FUNCTION_BLOCK SFC4 (* Basic Function Block Type *)
  (* Standard: 61499-2 *)
  (* Version 0.2, 2003-12-04, JHC, Rockwell Automation, Renamed for better indexing. *)
  (* Version 0.1, 2002-11-05, JHC, Rockwell Automation, Corrected missing ST element in Algorithm REQ. *)
  (* Version 0.0, 2000-05-30, JHC, Rockwell Automation *)
  (* Compiler header: package fb.rt.pnp; *)
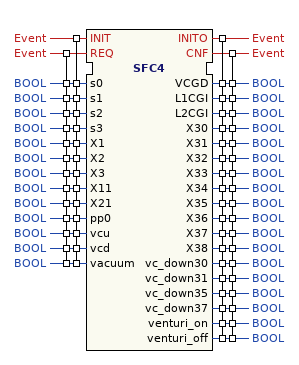
  EVENT_INPUT
    INIT WITH s0, s0, s0, s1, s2, s3, X1, X2, X3, X11, X21, pp0, vcu, vcd, vacuum; (* Initialization Request *)
    REQ WITH s0, s0, s1, s2, s3, X1, X2, X3, X11, X21, pp0, vcu, vcd, vacuum; (* Normal Execution Request *)
  END_EVENT
  EVENT_OUTPUT
    INITO WITH VCGD, L1CGI, L2CGI, X30, X30, X31, X32, X33, X34, X35, X36, X37, X38, vc_down30, vc_down31, vc_down35, vc_down37, venturi_on, venturi_off; (* Initialization Confirm *)
    CNF WITH VCGD, L1CGI, L2CGI, X30, X30, X31, X32, X33, X34, X35, X36, X37, X38, vc_down30, vc_down31, vc_down35, vc_down37, venturi_on, venturi_off; (* Execution Confirmation *)
  END_EVENT
  VAR_INPUT
    s0 : BOOL; (* Input event qualifier *)
    s1 : BOOL; (* Input event qualifier *)
    s2 : BOOL; (* Input event qualifier *)
    s3 : BOOL; (* Input event qualifier *)
    X1 : BOOL; (* Input event qualifier *)
    X2 : BOOL; (* Input event qualifier *)
    X3 : BOOL; (* Input event qualifier *)
    X11 : BOOL; (* Input event qualifier *)
    X21 : BOOL; (* Input event qualifier *)
    pp0 : BOOL; (* Input event qualifier *)
    vcu : BOOL; (* Input event qualifier *)
    vcd : BOOL; (* Input event qualifier *)
    vacuum : BOOL;
  END_VAR
  VAR_OUTPUT
    VCGD : BOOL; (* Output event qualifier *)
    L1CGI : BOOL;
    L2CGI : BOOL;
    X30 : BOOL;
    X31 : BOOL;
    X32 : BOOL;
    X33 : BOOL;
    X34 : BOOL;
    X35 : BOOL;
    X36 : BOOL;
    X37 : BOOL;
    X38 : BOOL;
    vc_down30 : BOOL;
    vc_down31 : BOOL;
    vc_down35 : BOOL;
    vc_down37 : BOOL;
    venturi_on : BOOL;
    venturi_off : BOOL;
  END_VAR
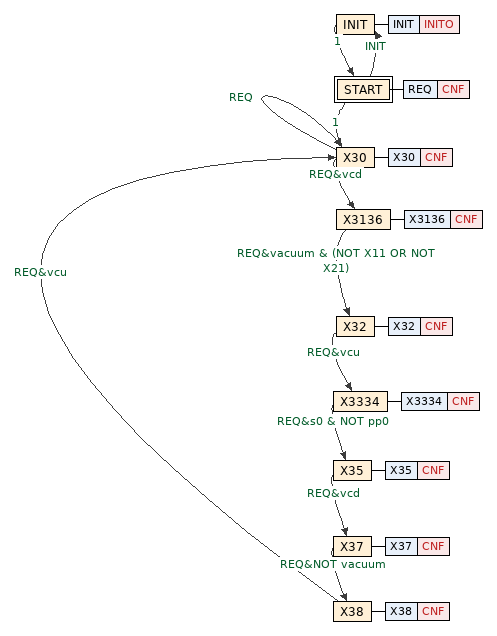
  EC_STATES
    START : REQ -> CNF; (* Initial State *)
    INIT : INIT -> INITO; (* Initialization *)
    X3136 : X3136 -> CNF; (* Normal execution *)
    X32 : X32 -> CNF;
    X3334 : X3334 -> CNF;
    X35 : X35 -> CNF;
    X37 : X37 -> CNF;
    X38 : X38 -> CNF;
    X30 : X30 -> CNF;
  END_STATES
  EC_TRANSITIONS
    START TO INIT := INIT;
    INIT TO START := 1;
    X3136 TO X32 := REQ&vacuum & (NOT X11 OR NOT X21);
    X32 TO X3334 := REQ&vcu;
    X3334 TO X35 := REQ&s0 & NOT pp0;
    X35 TO X37 := REQ&vcd;
    X37 TO X38 := REQ&NOT vacuum;
    X30 TO X3136 := REQ&vcd;
    X38 TO X30 := REQ&vcu;
    START TO X30 := 1;
    X30 TO X30 := REQ;
  END_TRANSITIONS
  ALGORITHM INIT IN ST: (* Initialization algorithm *)
X30:=true;
VCGD:=false;
L2CGI:=false;
L1CGI:=false;
X31:=false;
X32:=false;
X33:=false;
X34:=false;
X35:=false;
X36:=false;
X37:=false;
X38:=false;
vc_down30:=false;
vc_down31:=false;
vc_down35:=false;
vc_down37:=false;
venturi_on:=false;
venturi_off:=false;
System.out.println("SFC4: INIT");
  END_ALGORITHM
  ALGORITHM REQ IN Java: (* Normally executed algorithm *)
X38.value=false;
X30.value=true;
//System.out.println(s0.value + " " + s1.value + " " + s2.value + " " + s3.value + " " + X11.value + " " + X21.value);
  END_ALGORITHM
  ALGORITHM X30 IN ST:
X30:=true;
X38:=false;
IF (((s1 & X1) OR (s2 & X2) OR (s3 & X3)) & (NOT X11 OR NOT X21)) THEN
VCGD:= true;
vc_down30:=true;
END_IF
venturi_off:=false;
  END_ALGORITHM
  ALGORITHM X3136 IN ST:
venturi_on:=true;
vc_down30:=false;
vc_down31:=true;
X30:=false;
vc_down31:=true;
X31:=true;
X36:=true;
System.out.println("SFC4: X3136");
  END_ALGORITHM
  ALGORITHM X32 IN ST:
VCGD:=false;
X32:=true;
vc_down31:=false;
X31:=false;
X36:=true;
System.out.println("SFC4: X32");
  END_ALGORITHM
  ALGORITHM X3334 IN ST:
L1CGI:=true;
L2CGI:=true;
vc_down31:=false;
X32:=false;
X36:=true;
X33:=true;
X34:=true;
System.out.println("SFC4: X3334");
  END_ALGORITHM
  ALGORITHM X35 IN ST:
VCGD:=true;
L2CGI:=false;
L1CGI:=false;
vc_down35:=true;
X36:=true;
X33:=false;
X34:=false;
X35:=true;
System.out.println("SFC4: X35");
  END_ALGORITHM
  ALGORITHM X37 IN ST:
venturi_on:=false;
venturi_off:=true;
vc_down37:=true;
vc_down35:=false;
X36:=false;
X35:=false;
X37:=true;
System.out.println("SFC4: X37");
  END_ALGORITHM
  ALGORITHM X38 IN ST:
VCGD:=false;
vc_down37:=false;
X37:=false;
X38:=true;
System.out.println("SFC4: X38");
  END_ALGORITHM
END_FUNCTION_BLOCK
